{attribute 'qualified_only'}
VAR_GLOBAL
END_VAR

(* stored: Version 1.1.0.1, ProductVersion 3.1.4022.7
   GVL GVL_05_Manual_Test: Id {7fc7e54f-04b7-4b4a-96bf-46e5a410f39a} *)
